{attribute 'qualified_only'}
VAR_GLOBAL
    g_fbHoneyFill : FB_HoneyFill;
    g_fbSodaFill  : FB_SodaFill;
    g_fbWaterFill : FB_WaterFill;
END_VAR

(* stored: Version 1.1.0.1, ProductVersion 3.1.4024.16
   GVL GVL_References: Id {ab88abfe-d6b4-4773-85e4-b59f56500b94} *)
